// TIA Portal V20 export
TYPE "typeSequenceControlNodeHomeCheck_topTapeLoading"
// stored: Namespace Unit1.Em3
   STRUCT
      TapeLoadReq { ExternalWritable := 'False'} : Bool;
      TapeLoaded { ExternalWritable := 'False'} : Bool;
   END_STRUCT;
END_TYPE
